PROGRAM MAIN
VAR
	nAlive: INT;
	breset: BOOL;
	nDemoVariable : INT;
	nCX8200_State	AT %I*	: UINT;
END_VAR

VAR PERSISTENT
	nDemoVar_Persist: INT;
END_VAR

nAlive:= nAlive + 1;
GVL_AHDataModbus.nCX8200_State_MB := nCX8200_State;

P_SystemDK.M_nCyclic(bReset := breset );
P_DALI_DIAG();
DALI_Commissioning();
P_DALI_Energy_Line();
P_AHModbusComm();
P_DALI_Background();

//Gange
P_Gang_2_143A();
P_Gang_3_159A();
P_Gang_3_157();
P_Gang_7_153();
P_Rum_2_135();
P_Gang_Atrium();
//P_Gang_atrium();



//FoldeDøre
//P_Foldedoer_5_125();

//Rum
P_Rum_2_145();
P_Rum_3_155();
P_Rum_3_157A();
P_Rum_3_155();

//Trapper
P_Trappe_T2();
P_Trappe_T3();
//Testprogrammer
//P_DALI_Energy_Firmware_Test();

END_PROGRAM

(* stored: Version 1.1.0.1
   POU MAIN: Id {6bf17237-b1a6-4c57-bf47-1238f1ca1a56}, SpecialFunc None *)
